{attribute 'linkalways'} 
{attribute 'no_explicit_call' := 'This FB is a CLASS and must be accessed using methods or properties'}
{attribute 'enable_dynamic_creation'}
FUNCTION_BLOCK FINAL SUB_DWORD EXTENDS Node
VAR
	in1 : _DWORD(0);
	in2 : _DWORD(0);
	out : _DWORD(0);
END_VAR

METHOD PUBLIC Clone : I_Node
VAR
	pNode : POINTER TO SUB_DWORD;
END_VAR
pNode := __NEW(SUB_DWORD);
Clone := pNode^;
END_METHOD

METHOD FB_init : BOOL
VAR_INPUT
	bInitRetains : BOOL; // if TRUE, the retain variables are initialized (warm start / cold start)
	bInCopyCode : BOOL;  // if TRUE, the instance afterwards gets moved into the copy code (online change)
END_VAR
AddInput('in1',THIS^.in1);
AddInput('in2',THIS^.in2);
AddOutput('out', THIS^.out);
END_METHOD

METHOD PROTECTED OnExecute
VAR
END_VAR
out.Value := in1.Value - in2.Value;
END_METHOD

END_FUNCTION_BLOCK

(* stored: Version 1.1.0.1, ProductVersion 3.1.4024.15
   POU SUB_DWORD: Id {31ddd61b-6d95-41e7-9261-782e7b9621c6}, SpecialFunc None
   Folder Constructor: Id {71539be3-6203-4169-973d-7fc84f695ac6}
   Method Clone: Id {2e0d65ea-6a46-4685-9045-dc9ecef81b5e}
   Method FB_init: Id {4958c549-cc7b-41f6-b69d-630c2514fcf1}
   Method OnExecute: Id {433f1a99-df7a-4523-8c78-3c480f718d6a} *)
